// TIA Portal V20 export
FUNCTION_BLOCK "05 T4 LANT Sequence"   // FB1512, GRAPH
// stored: AutoNumber false, GraphVersion 6.0, InitialValuesAcquisition false, SetENOAutomatically false
   // inherited from GRAPH_BASE
   VAR_INPUT
      OFF_SQ : Bool := false;
      INIT_SQ : Bool := false;
      ACK_EF : Bool := false;
      S_PREV : Bool := false;
      S_NEXT : Bool := false;
      SW_AUTO : Bool := false;
      SW_TAP : Bool := false;
      SW_TOP : Bool := false;
      SW_MAN : Bool := false;
      S_SEL : Int := 0;
      S_ON : Bool := false;
      S_OFF : Bool := false;
      T_PUSH : Bool := false;
   END_VAR
   VAR_OUTPUT
      S_NO : Int := 0;
      S_MORE : Bool := false;
      S_ACTIVE : Bool := false;
      ERR_FLT : Bool := false;
      AUTO_ON : Bool := false;
      TAP_ON : Bool := false;
      TOP_ON : Bool := false;
      MAN_ON : Bool := false;
   END_VAR
BEGIN
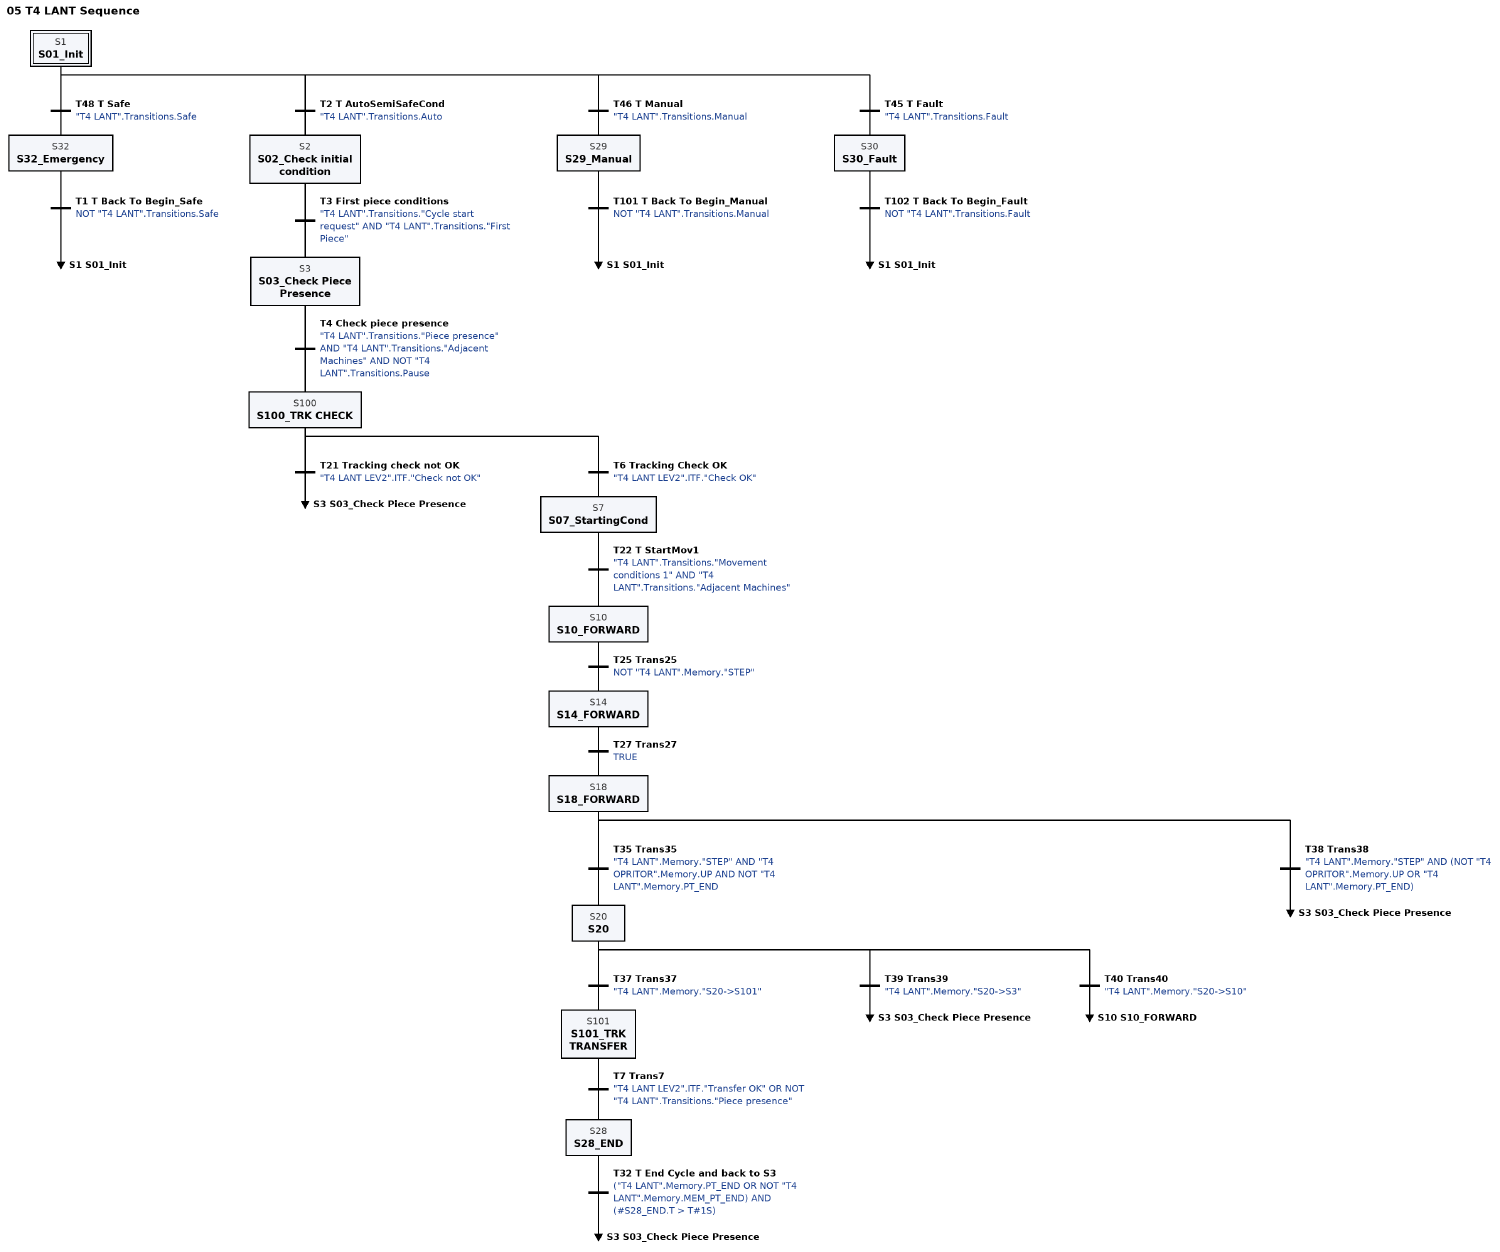
   // permanent pre-instructions
   NETWORK 1
      "01 T4 LANT Alarms"();
   NETWORK 2
      "02 T4 LANT HMI"();
   NETWORK 3
      "03 T4 LANT Aux"();
   NETWORK 4
      "04 T4 LANT Transitions"();

   // sequencer 1
   INITIAL_STEP S01_Init:   // S1, max time T#10S, warning time T#7S
   END_STEP
   TRANSITION "T Safe" FROM S01_Init TO S32_Emergency   // T48
      := "T4 LANT".Transitions.Safe;
   END_TRANSITION
   TRANSITION "T AutoSemiSafeCond" FROM S01_Init TO "S02_Check initial condition"   // T2
      := "T4 LANT".Transitions.Auto;
   END_TRANSITION
   TRANSITION "T Manual" FROM S01_Init TO S29_Manual   // T46
      := "T4 LANT".Transitions.Manual;
   END_TRANSITION
   TRANSITION "T Fault" FROM S01_Init TO S30_Fault   // T45
      := "T4 LANT".Transitions.Fault;
   END_TRANSITION
   STEP "S03_Check Piece Presence":   // S3, max time T#10S, warning time T#7S
   END_STEP
   TRANSITION "Check piece presence" FROM "S03_Check Piece Presence" TO "S100_TRK CHECK"   // T4
      := "T4 LANT".Transitions."Piece presence" AND "T4 LANT".Transitions."Adjacent Machines" AND NOT "T4 LANT".Transitions.Pause;
   END_TRANSITION
   STEP S32_Emergency:   // S32, max time T#10S, warning time T#7S
   END_STEP
   TRANSITION "T Back To Begin_Safe" FROM S32_Emergency TO S01_Init   // T1, jump
      := NOT "T4 LANT".Transitions.Safe;
   END_TRANSITION
   STEP S29_Manual:   // S29, max time T#10S, warning time T#7S
   END_STEP
   TRANSITION "T Back To Begin_Manual" FROM S29_Manual TO S01_Init   // T101, jump
      := NOT "T4 LANT".Transitions.Manual;
   END_TRANSITION
   STEP "S02_Check initial condition":   // S2, max time T#10S, warning time T#7S
   END_STEP
   TRANSITION "First piece conditions" FROM "S02_Check initial condition" TO "S03_Check Piece Presence"   // T3
      := "T4 LANT".Transitions."Cycle start request" AND "T4 LANT".Transitions."First Piece";
   END_TRANSITION
   STEP S30_Fault:   // S30, max time T#10S, warning time T#7S
   END_STEP
   TRANSITION "T Back To Begin_Fault" FROM S30_Fault TO S01_Init   // T102, jump
      := NOT "T4 LANT".Transitions.Fault;
   END_TRANSITION
   STEP S28_END:   // S28, max time T#10S, warning time T#7S
   END_STEP
   TRANSITION "T End Cycle and back to S3" FROM S28_END TO "S03_Check Piece Presence"   // T32, jump: Assenza pezzo o ok da robot
      := ("T4 LANT".Memory.PT_END OR NOT "T4 LANT".Memory.MEM_PT_END) AND (#S28_END.T > T#1S);
   END_TRANSITION
   STEP S10_FORWARD:   // S10, max time T#10S, warning time T#7S
   END_STEP
   TRANSITION Trans25 FROM S10_FORWARD TO S14_FORWARD   // T25
      := NOT "T4 LANT".Memory."STEP";
   END_TRANSITION
   STEP S14_FORWARD:   // S14, max time T#10S, warning time T#7S
   END_STEP
   TRANSITION Trans27 FROM S14_FORWARD TO S18_FORWARD   // T27
      := TRUE;
   END_TRANSITION
   STEP S18_FORWARD:   // S18, max time T#10S, warning time T#7S
   END_STEP
   TRANSITION Trans35 FROM S18_FORWARD TO S20   // T35
      := "T4 LANT".Memory."STEP" AND "T4 OPRITOR".Memory.UP AND NOT "T4 LANT".Memory.PT_END;
   END_TRANSITION
   TRANSITION Trans38 FROM S18_FORWARD TO "S03_Check Piece Presence"   // T38, jump
      := "T4 LANT".Memory."STEP" AND (NOT "T4 OPRITOR".Memory.UP OR "T4 LANT".Memory.PT_END);
   END_TRANSITION
   STEP "S100_TRK CHECK":   // S100, max time T#10S, warning time T#7S
   END_STEP
   TRANSITION "Tracking check not OK" FROM "S100_TRK CHECK" TO "S03_Check Piece Presence"   // T21, jump
      := "T4 LANT LEV2".ITF."Check not OK";
   END_TRANSITION
   TRANSITION "Tracking Check OK" FROM "S100_TRK CHECK" TO S07_StartingCond   // T6
      := "T4 LANT LEV2".ITF."Check OK";
   END_TRANSITION
   STEP "S101_TRK TRANSFER":   // S101, max time T#10S, warning time T#7S
   END_STEP
   TRANSITION Trans7 FROM "S101_TRK TRANSFER" TO S28_END   // T7
      := "T4 LANT LEV2".ITF."Transfer OK" OR NOT "T4 LANT".Transitions."Piece presence";
   END_TRANSITION
   STEP S07_StartingCond:   // S7, max time T#10S, warning time T#7S
   END_STEP
   TRANSITION "T StartMov1" FROM S07_StartingCond TO S10_FORWARD   // T22
      := "T4 LANT".Transitions."Movement conditions 1" AND "T4 LANT".Transitions."Adjacent Machines";
   END_TRANSITION
   STEP S20:   // S20, max time T#10S, warning time T#7S
   END_STEP
   TRANSITION Trans37 FROM S20 TO "S101_TRK TRANSFER"   // T37
      := "T4 LANT".Memory."S20->S101";
   END_TRANSITION
   TRANSITION Trans39 FROM S20 TO "S03_Check Piece Presence"   // T39, jump
      := "T4 LANT".Memory."S20->S3";
   END_TRANSITION
   TRANSITION Trans40 FROM S20 TO S10_FORWARD   // T40, jump
      := "T4 LANT".Memory."S20->S10";
   END_TRANSITION

   // permanent post-instructions
   NETWORK 1
      "06 T4 LANT Output"();
   NETWORK 2
      "07 T4 LANT LEV2"();
END_FUNCTION_BLOCK
